(* Schneider Machine Expert - Basic project Yeni proje33, file version 1.8.0.0 *)
(* ProjectInformations: Name=Yeni proje *)

HARDWARE
  Cpu 0: TM221ME16T/G
  ModuleExtensionObject 0: TM3DI8/G
  ModuleExtensionObject 1: TM3AQ2/G
  EthernetConfiguration: NetworkName=M221, IpAllocationMode=FixedAddress, IpAddress=192.168.0.15, SubnetMask=255.255.255.0
  SerialLineConfiguration: Baud=Baud19200, Parity=ParityNone, DataBits=DataBits8, StopBits=StopBits1, PhysicalMedium=PhysicalMediumRs485, TransmissionMode=TransmissionModeModbusRtu, SlaveId=1, Addressing=SlaveAddressing
  MastTask: UsePeriodScanMode=false, PeriodScan=100
  FastTask: Period=255
  CpuBehavior: StartingMode=StartAsPreviousState, AutoSaveRamOnEeprom=true, WatchdogPeriod=250

SYMBOLS  (address, symbol, comment, settings)
  %M0         "HMI/FIRÇA YUKARI"
  %M1         "HMI/FIRÇA AŞAĞI"
  %M2         "HMI/FIRÇA 2 YUKARI"
  %M3         "HMI/FIRÇA 2 AŞAĞI"
  %M4         "HMI BANT START"
  %M5         "HMI OSILASYON START"
  %M6         "427"
  %M7         "428"
  %I0.0       "403/FIRÇA1 ÜST SINIR ANAHTARI"
  %I0.1       "402/FIRÇA1 ALT SINIR ANAHTARI"
  %I0.2       "405/FIRÇA2/ÜST SINIR ANAHTARI"
  %I0.3       "404/FIRÇA2/ ALT SINIR ANAHTARI"
  %Q0.0       "421/FIRÇA YUKARI"
  %Q0.1       "422/FIRÇA AŞAĞI"
  %Q0.2       "423/FIRÇA 2 YUKARI"
  %Q0.3       "424/FIRÇA 2 AŞAĞI"
  %Q0.4       "425/BANT START"
  %Q0.5       "426/OSILASYON START"
  %Q0.6       "427"
  %Q0.7       "428"

POU Yeni POU
  (* SectionNumber=1 *)

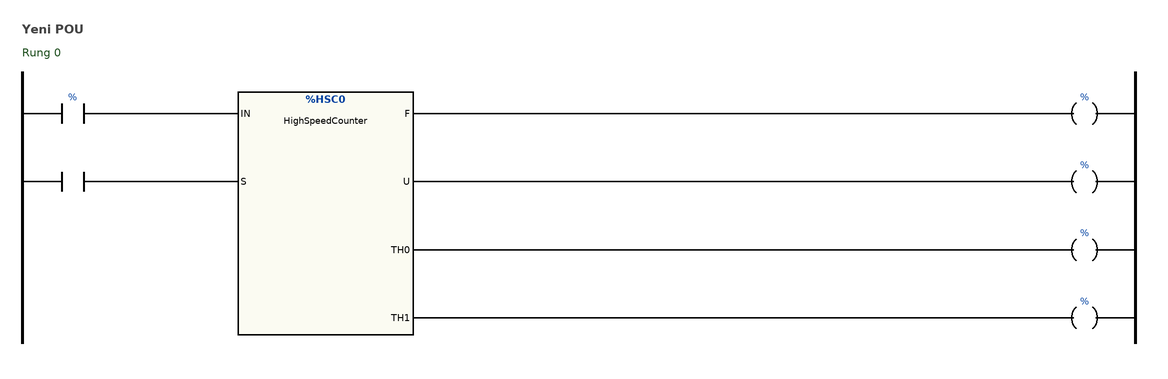

// Rung 0
  (* no IL stored for this rung *)
